Fanuc KAREL source: kb00083.KL

-- PROVISIONAL review KL for V770-1; original PC SHA256 3889422cbfcde47e4aab22905667e99453e06d5ebf707ecb30aa4647fe3269e8
-- Incomplete behavior may be omitted. Consult companion uncertainty JSON. Do not deploy.
PROGRAM KB00083
%NOLOCKGROUP
BEGIN
  -- UNRESOLVED_PC offsets 5-12; opcodes 9D,23
  -- UNRESOLVED_PC offsets 17-24; opcodes 9D,23
  -- UNRESOLVED_PC offsets 29-36; opcodes 9D,23
  -- UNRESOLVED_PC offsets 41-48; opcodes 9D,23
  -- UNRESOLVED_PC offsets 53-81; opcodes 27,22,22,22,22,31
  -- UNRESOLVED_PC offsets 86-90; opcodes 7F
END KB00083
